// TIA Portal V19 export
TYPE "C104_VAR_IF_NSI_TYPIC"
   STRUCT
      BSC1 { ExternalAccessible := 'False'; ExternalVisible := 'False'; ExternalWritable := 'False'} : Bool;   // Noodstroominstallatie beschikbaar
      BSC2 { ExternalAccessible := 'False'; ExternalVisible := 'False'; ExternalWritable := 'False'} : Bool;   // Noodstroominstallatie niet beschikbaar
      BSC3 { ExternalAccessible := 'False'; ExternalVisible := 'False'; ExternalWritable := 'False'} : Bool;   // Noodstroominstallatie beperkt beschikbaar
      ENE_TOT { ExternalAccessible := 'False'; ExternalVisible := 'False'; ExternalWritable := 'False'} : Real;   // Totaal energieverbruik noodstroominstallatie
   END_STRUCT;
END_TYPE
